// TwinCAT 3 PLC project Decorator_Pattern
// ProgramVersion: 3.1.4024.0
// libraries:
//   Tc2_Standard, * (Beckhoff Automation GmbH)
//   Tc2_System, * (Beckhoff Automation GmbH)
//   Tc3_Module, * (Beckhoff Automation GmbH)
// project tree:
//   Analogues/ AnalogueTerminal.TcPOU, ITF_Analogue.TcIO
//   Decorators/ DecimationDecorator.TcPOU, DecoratorBase.TcPOU, OffsetDecorator.TcPOU, ScaleDecorator.TcPOU
//   / PlcTask.TcTTO
//   POUs/ MAIN.TcPOU
// (motion and I/O tree: see PLC project simple_factory_pattern)
// real-time tasks:
//   TASK PlcTask: cycle T#10ms, priority 20, ADS port 350
//   TASK PlcTask1: cycle T#10ms, priority 21, ADS port 351
//   TASK PlcTask2: cycle T#10ms, priority 22, ADS port 352
//   TASK PlcTask3: cycle T#10ms, priority 23, ADS port 353
//   TASK PlcTask4: cycle T#10ms, priority 24, ADS port 354
//   TASK PlcTask5: cycle T#10ms, priority 25, ADS port 355
//   TASK PlcTask6: cycle T#10ms, priority 26, ADS port 356
//   TASK PlcTask7: cycle T#10ms, priority 27, ADS port 357
//   TASK PlcTask8: cycle T#10ms, priority 28, ADS port 358
//   TASK PlcTask9: cycle T#10ms, priority 29, ADS port 359
//   TASK PlcTask10: cycle T#10ms, priority 30, ADS port 360
//   TASK PlcTask11: cycle T#10ms, priority 31, ADS port 361

CONFIGURATION Decorator_Pattern
    RESOURCE PLC ON TwinCAT3
        TASK PlcTask(INTERVAL := T#10ms, PRIORITY := 26);
        PROGRAM MAIN WITH PlcTask : MAIN;
    END_RESOURCE
END_CONFIGURATION

// ---- Analogues/ITF_Analogue.TcIO
INTERFACE ITF_Analogue

METHOD GetValue : LREAL
VAR_INPUT
END_VAR
END_METHOD

END_INTERFACE

// ---- POUs/MAIN.TcPOU
PROGRAM MAIN
VAR
	MyAnalogueTerminal : AnalogueTerminal;
	SignalDecimation : DecimationDecorator;
	SignalOffset : OffsetDecorator;
	SignalScale : ScaleDecorator;
	AnalogueChannel : ITF_Analogue;
	init: BOOL;
	MySignal: LREAL;
END_VAR

IF NOT init	THEN
	init := TRUE;
	SignalDecimation.MyWrappee := MyAnalogueTerminal;
	SignalScale.MyWrappee := SignalDecimation;
	SignalOffset.MyWrappee := SignalScale;
	AnalogueChannel := SignalOffset;
ELSE
	MySignal := AnalogueChannel.GetValue();
END_IF

END_PROGRAM

// ---- Analogues/AnalogueTerminal.TcPOU
FUNCTION_BLOCK AnalogueTerminal IMPLEMENTS ITF_Analogue
VAR
	_SomeValueFromIO : INT := 8192;
END_VAR

METHOD GetValue : LREAL
VAR_INPUT
END_VAR
GetValue :=  (_SomeValueFromIO/32767.0)*10.0;
END_METHOD

END_FUNCTION_BLOCK

// ---- Decorators/DecimationDecorator.TcPOU
FUNCTION_BLOCK DecimationDecorator EXTENDS DecoratorBase
VAR
	decimationfactor : INT := 1;
	currentValue: LREAL;
END_VAR

METHOD GetValue : lreal
IF (THIS^.wrappee <> 0) THEN
	IF decimationfactor = 5 THEN
		GetValue := THIS^.wrappee.GetValue();
		currentValue := GetValue;
		decimationfactor := 1;
	ELSE
		decimationfactor := decimationfactor + 1;
		GetValue := currentValue;
	END_IF
END_IF
END_METHOD

END_FUNCTION_BLOCK

// ---- Decorators/DecoratorBase.TcPOU
FUNCTION_BLOCK DecoratorBase IMPLEMENTS ITF_Analogue
VAR
	wrappee : ITF_Analogue;
END_VAR

METHOD GetValue : LREAL
END_METHOD

PROPERTY MyWrappee : itf_analogue
GET
MyWrappee := wrappee;
END_GET
SET
wrappee := MyWrappee;
END_SET
END_PROPERTY

END_FUNCTION_BLOCK

// ---- Decorators/OffsetDecorator.TcPOU
FUNCTION_BLOCK OffsetDecorator EXTENDS DecoratorBase
VAR
END_VAR

METHOD GetValue : lreal
IF (THIS^.wrappee <> 0) THEN
 	GetValue := THIS^.wrappee.GetValue() - 10.0;
END_IF
END_METHOD

END_FUNCTION_BLOCK

// ---- Decorators/ScaleDecorator.TcPOU
FUNCTION_BLOCK ScaleDecorator EXTENDS DecoratorBase
VAR
END_VAR

METHOD GetValue : LREAL
IF (THIS^.wrappee <> 0) THEN
  GetValue := (THIS^.wrappee.GetValue()/20.0)*100.0;
END_IF
END_METHOD

END_FUNCTION_BLOCK
